FUNCTION_BLOCK FB_SIM_SA_CHANNEL
VAR_INPUT
END_VAR
VAR_OUTPUT
END_VAR
VAR
	cfg:	T_SA_SIM_CH_CFG;
	ctrl:	T_SA_SIM_CH_CTRL;
	stat:	T_SA_SIM_CH_STATUS;
	
	fbTimer:		TON;

END_VAR

// Execute State Machine
M_StateMachine();

METHOD M_GetChSimReply : STRING(255)
VAR_INPUT
	{attribute 'OPC.UA.DA' := '0'}
	in_sCmd:	STRING(255);		// String received from a client
END_VAR
VAR
	sReply:	STRING(255);
	sTmp:	STRING;
	lrVal:	LREAL;
	nValue:	UINT;
	i:		INT;
    fbFormat   : FB_FormatString;
    sOut       : T_MaxString;
	nCh:	INT := 8;	// Number of channels for models 218 and 224
END_VAR

IF FIND (in_sCmd, '?') > 0 THEN
	// This is a query command.
	// There is a reply.
	// Check commands one by one.

	IF FIND (in_sCmd, 'STAT?') > 0 THEN
		// Channel state
		M_GetChSimReply	:= UDINT_TO_STRING(stat.nSTATE);
	ELSIF FIND (in_sCmd, 'CAL:OPT?') > 0 THEN
		// Channel state
		M_GetChSimReply	:= UINT_TO_STRING(cfg.nCAL_OPT);
	ELSIF FIND (in_sCmd, 'REF:OPT?') > 0 THEN
		// Channel state
		M_GetChSimReply	:= UINT_TO_STRING(cfg.nREF_OPT);
	ELSIF FIND (in_sCmd, 'PCON:OPT?') > 0 THEN
		// Channel Positioner control otions
		M_GetChSimReply	:= UINT_TO_STRING(cfg.nPCON_OPT);
	ELSIF FIND (in_sCmd, 'INP:THR?') > 0 THEN
		// Channel in-position threshold
		M_GetChSimReply	:= UDINT_TO_STRING(cfg.nINP_THR);
	ELSIF FIND (in_sCmd, 'INP:DEL?') > 0 THEN
		// Channel in-position delay
		M_GetChSimReply	:= UDINT_TO_STRING(cfg.nINP_DEL);
	ELSIF FIND (in_sCmd, 'RLIM:MIN?') > 0 THEN
		// Channel Limit Min
		M_GetChSimReply	:= LINT_TO_STRING(cfg.lnRLIM_MIN);
	ELSIF FIND (in_sCmd, 'RLIM:MAX?') > 0 THEN
		// Channel Limit Max
		M_GetChSimReply	:= LINT_TO_STRING(cfg.lnRLIM_MAX);
	ELSIF FIND (in_sCmd, 'POS:TARG?') > 0 THEN
		// Channel target position
		M_GetChSimReply	:= LINT_TO_STRING(stat.lnPosTarget);
	ELSIF FIND (in_sCmd, 'POS:CURR?') > 0 THEN
		// Channel actual position
		M_GetChSimReply	:= LINT_TO_STRING(stat.lnPosActual);
	ELSIF FIND (in_sCmd, 'CLIN?') > 0 THEN
		// Channel 
		M_GetChSimReply	:= DINT_TO_STRING(cfg.nCLIN);
	ELSIF FIND (in_sCmd, 'TUN:BASE:UNIT?') > 0 THEN
		// Channel 
		M_GetChSimReply	:= DINT_TO_STRING(cfg.nBASE_UNIT);
	ELSIF FIND (in_sCmd, 'TUN:BASE:RES?') > 0 THEN
		// Channel 
		M_GetChSimReply	:= DINT_TO_STRING(cfg.nBASE_RES);
	ELSIF FIND (in_sCmd, 'TUN:MTYP?') > 0 THEN
		// Channel 
		M_GetChSimReply	:= DINT_TO_STRING(cfg.nTUN_MTYP);
	ELSIF FIND (in_sCmd, 'TUN:RTYP?') > 0 THEN
		// Channel 
		M_GetChSimReply	:= LINT_TO_STRING(cfg.nTUN_RTYP);
	END_IF
ELSE
	// This is a control command.
	// There is NO reply.
	// BUT there are some action to be taken

	IF FIND (in_sCmd, 'CAL:OPT ') > 0 THEN
		// Get the value
		sTmp			:= DELETE(in_sCmd,8,1);
		cfg.nCAL_OPT	:= STRING_TO_UINT(sTmp);
	ELSIF FIND (in_sCmd, 'REF:OPT ') > 0 THEN
		// Get the value
		sTmp			:= DELETE(in_sCmd,8,1);
		cfg.nREF_OPT	:= STRING_TO_UINT(sTmp);
	ELSIF FIND (in_sCmd, 'PCON:OPT ') > 0 THEN
		// Get the value
		sTmp			:= DELETE(in_sCmd,9,1);
		cfg.nPCON_OPT	:= STRING_TO_UINT(sTmp);
	ELSIF FIND (in_sCmd, 'INP:THR ') > 0 THEN
		// Get the value
		sTmp			:= DELETE(in_sCmd,8,1);
		cfg.nINP_THR	:= STRING_TO_UDINT(sTmp);
	ELSIF FIND (in_sCmd, 'INP:DEL ') > 0 THEN
		// Get the value
		sTmp			:= DELETE(in_sCmd,8,1);
		cfg.nINP_DEL	:= STRING_TO_UDINT(sTmp);
	ELSIF FIND (in_sCmd, 'RLIM:MIN ') > 0 THEN
		// Get the value
		sTmp			:= DELETE(in_sCmd,9,1);
		cfg.lnRLIM_MIN	:= STRING_TO_UINT(sTmp);
	ELSIF FIND (in_sCmd, 'RLIM:MAX ') > 0 THEN
		// Get the value
		sTmp			:= DELETE(in_sCmd,9,1);
		cfg.lnRLIM_MAX	:= STRING_TO_UINT(sTmp);
	ELSIF FIND (in_sCmd, 'POS:TARG ') > 0 THEN
		// Get the value
		sTmp			:= DELETE(in_sCmd,9,1);
		stat.lnPosTarget:= F_STRING_TO_LINT(sTmp);
	ELSIF FIND (in_sCmd, 'POS:CURR ') > 0 THEN
		// Get the value
		sTmp			:= DELETE(in_sCmd,9,1);
		stat.lnPosActual:= F_STRING_TO_LINT(sTmp);
	ELSIF FIND (in_sCmd, 'VEL ') > 0 THEN
		// Get the value
		sTmp			:= DELETE(in_sCmd,4,1);
		cfg.lnVEL		:= F_STRING_TO_LINT(sTmp);
		ctrl.lnVEL		:= F_STRING_TO_LINT(sTmp);
	ELSIF FIND (in_sCmd, 'POS ') > 0 THEN
		// Get the value
		sTmp			:= DELETE(in_sCmd,4,1);
		stat.lnPosActual:= F_STRING_TO_LINT(sTmp);
	END_IF
	
	// There is no reply to control commands !!!
	M_GetChSimReply	:= '';
END_IF
END_METHOD

METHOD M_StartCAL
VAR_INPUT
END_VAR
// Start CALibration simulation
;
END_METHOD

METHOD M_StartMOVE
VAR_INPUT
	in_lnPos:	LINT;	// Target Position
	in_lnVel:	LINT;	// Target Velocity
END_VAR
VAR 
	nState:		UDINT := 0;
	nTime:		UDINT :=0;	// Calculated move time [ms].
END_VAR
// Start MOVE simulation

// Set target velocity and position.
ctrl.lnVEL			:= in_lnVel;
ctrl.lnPOS			:= in_lnPos;
stat.lnPosTarget	:= in_lnPos;
stat.lnPosStart		:= stat.lnPosActual;	// MOVE started from this position

// Get the distance to move.
// If distance is zero, do nothing.
stat.lnDistance	:= ctrl.lnPOS - stat.lnPosActual;
IF stat.lnDistance = 0	THEN
	// No movement
	fbTimer(IN:=FALSE);
	RETURN;
END_IF

nState	:= nState OR E_SA_CH_STATE.BIT_ACTIVELY_MOVING;
nState	:= nState OR E_SA_CH_STATE.BIT_CLOSED_LOOP_ACTIVE;
nState	:= nState OR E_SA_CH_STATE.BIT_SENSOR_PRESENT;
nState	:= nState OR E_SA_CH_STATE.BIT_IS_CALIBRATED;
nState	:= nState OR E_SA_CH_STATE.BIT_IS_REFERENCED;
nState	:= nState OR E_SA_CH_STATE.BIT_AMPLIFIER_ENABLED;

stat.nSTATE	:= nState;

// Get time [ms] needed for the move
IF in_lnVel = 0	THEN
	nTime	:= 1000;
ELSE	
	nTime	:= LINT_TO_UDINT(1000 * ABS(stat.lnDistance) / in_lnVel);
END_IF

IF nTime > 0 THEN
	// Set the positioner State Machine State
	stat.nPosState	:=	E_SA_POS_SM_STATE.MOVING;
	
	// Start the timer.
	// Simulated REFerencing should finish in 5 sec.
	fbTimer(IN:=FALSE);
	fbTimer(IN:=TRUE,PT:=UDINT_TO_TIME(nTime));
ELSE
	// No movement
	fbTimer(IN:=FALSE);
END_IF
END_METHOD

METHOD M_StartREF
VAR_INPUT
END_VAR
VAR 
	nState:		UDINT := 0;
END_VAR
// Start REFerencing simulation

nState	:= nState OR E_SA_CH_STATE.BIT_ACTIVELY_MOVING;
nState	:= nState OR E_SA_CH_STATE.BIT_CLOSED_LOOP_ACTIVE;
nState	:= nState OR E_SA_CH_STATE.BIT_REFERENCING;
nState	:= nState OR E_SA_CH_STATE.BIT_SENSOR_PRESENT;
nState	:= nState OR E_SA_CH_STATE.BIT_AMPLIFIER_ENABLED;

stat.nSTATE	:= nState;

// Set the positioner State Machine State
stat.nPosState	:=	E_SA_POS_SM_STATE.CALIB_REF;

// Start the timer.
// Simulated REFerencing should finish in 5 sec.
fbTimer(IN:=FALSE);
fbTimer(IN:=TRUE,PT:=T#5S);
END_METHOD

METHOD M_StateMachine
VAR_INPUT
END_VAR
VAR 
	nState:		UDINT := 0;
	lrProgress:	LREAL;		// Movement progress [0.0..1.0]
	lnPosInc:	LINT;		// Position increment from starting position.
END_VAR
// Execute the timer.
fbTimer();

CASE stat.nPosState OF
	E_SA_POS_SM_STATE.CALIB_REF:
		// Check if referencing is complete.
		IF fbTimer.Q THEN
			// Reset timer
			fbTimer(IN:=FALSE);
			// Set flags for completed REFerencing
			nState	:= nState OR E_SA_CH_STATE.BIT_CLOSED_LOOP_ACTIVE;
			nState	:= nState OR E_SA_CH_STATE.BIT_SENSOR_PRESENT;
			nState	:= nState OR E_SA_CH_STATE.BIT_IS_CALIBRATED;
			nState	:= nState OR E_SA_CH_STATE.BIT_IS_REFERENCED;
			nState	:= nState OR E_SA_CH_STATE.BIT_REFERENCE_MARK;
			nState	:= nState OR E_SA_CH_STATE.BIT_AMPLIFIER_ENABLED;
			nState	:= nState OR E_SA_CH_STATE.BIT_IN_POSITION;
			
			stat.nSTATE	:= nState;
			
			// Set the calibrated position
			stat.lnPosTarget	:= cfg.lnREF_POS;
			stat.lnPosActual	:= cfg.lnREF_POS;
			
			// Set the positioner State Machine State
			stat.nPosState	:=	E_SA_POS_SM_STATE.OP;
		END_IF
	E_SA_POS_SM_STATE.MOVING:
		// Simulate movement progress
		IF fbTimer.PT = T#0MS THEN
			RETURN;
		END_IF
		lrProgress	:= TIME_TO_LREAL(fbTimer.ET) / TIME_TO_LREAL(fbTimer.PT);
		lnPosInc	:= LREAL_TO_LINT(LINT_TO_LREAL(stat.lnDistance) * lrProgress);
		stat.lnPosActual	:= stat.lnPosStart + lnPosInc;
		
		// Check if the move is complete.
		IF fbTimer.Q THEN
			// Reset timer
			fbTimer(IN:=FALSE);
			// Set flags for completed REFerencing
			nState	:= nState OR E_SA_CH_STATE.BIT_CLOSED_LOOP_ACTIVE;
			nState	:= nState OR E_SA_CH_STATE.BIT_SENSOR_PRESENT;
			nState	:= nState OR E_SA_CH_STATE.BIT_IS_CALIBRATED;
			nState	:= nState OR E_SA_CH_STATE.BIT_IS_REFERENCED;
			nState	:= nState OR E_SA_CH_STATE.BIT_AMPLIFIER_ENABLED;
			nState	:= nState OR E_SA_CH_STATE.BIT_IN_POSITION;
			
			stat.nSTATE	:= nState;
			
			// Set the positioner State Machine State
			stat.nPosState	:=	E_SA_POS_SM_STATE.OP;
		END_IF
END_CASE
END_METHOD

METHOD M_STOP
VAR_INPUT
END_VAR
VAR 
	nState:		UDINT := 0;
END_VAR
// STOP MOVE simulation
// Start MOVE simulation

// No movement. Stop the timer.
fbTimer(IN:=FALSE);

nState	:= nState OR E_SA_CH_STATE.BIT_CLOSED_LOOP_ACTIVE;
nState	:= nState OR E_SA_CH_STATE.BIT_SENSOR_PRESENT;
nState	:= nState OR E_SA_CH_STATE.BIT_IS_CALIBRATED;
nState	:= nState OR E_SA_CH_STATE.BIT_IS_REFERENCED;
nState	:= nState or E_SA_CH_STATE.BIT_AMPLIFIER_ENABLED;

stat.nSTATE	:= nState;

stat.nPosState	:=	E_SA_POS_SM_STATE.OP;
END_METHOD

END_FUNCTION_BLOCK

(* stored: Version 1.1.0.1, ProductVersion 3.1.4024.10
   POU FB_SIM_SA_CHANNEL: Id {84d5a22a-8fbd-474a-92ad-3ec9d00e1a18}, SpecialFunc None
   Method M_GetChSimReply: Id {90494e50-17c0-43f1-97ab-c84ea9729b3e}
   Method M_StartCAL: Id {ce5cd431-a44b-4368-99ae-5503f9f284a5}
   Method M_StartMOVE: Id {9b92d063-b605-4251-8b3f-d34b573d095a}
   Method M_StartREF: Id {331d8561-6b8c-4e93-b808-11a785be6764}
   Method M_StateMachine: Id {2584681c-8189-424d-b208-9753c62b37fa}
   Method M_STOP: Id {a3b503df-f708-4e31-a191-0c056e34c1e0} *)
